FUNCTION_BLOCK FB_Stan_Held EXTENDS FB_SITP_Element
VAR

END_VAR

METHOD FB_init : BOOL
VAR_INPUT
	bInitRetains : BOOL; // if TRUE, the retain variables are initialized (warm start / cold start)
	bInCopyCode : BOOL;  // if TRUE, the instance afterwards gets moved into the copy code (online change)
END_VAR
THIS^.PrzypiszTekstDo (refstEtykieta := THIS^.stNazwa, eJezyk := B_Baza.E_Jezyki.pl, wsTekst	:= "Przerywanie");
THIS^.PrzypiszTekstDo (refstEtykieta := THIS^.stNazwa, eJezyk := B_Baza.E_Jezyki.de, wsTekst	:= "Abbruch");    
THIS^.PrzypiszTekstDo (refstEtykieta := THIS^.stNazwa, eJezyk := B_Baza.E_Jezyki.en, wsTekst	:= "Aborting");
END_METHOD

METHOD PUBLIC WywolajAkcjePBDlaStanu : BOOL
VAR_INPUT
	iNumerPB				: INT;
END_VAR
WywolajAkcjePBDlaStanu			:= THIS^.refstDaneSITP.refarrPB [iNumerPB].SP_Held ();
END_METHOD

(*			
	EVERDE sp. z o.o.
	Rafał Osajda		18.06.2025		TC 4024.66
	Zwraca true jak wyjście ze stanu jest możliwe
*)
METHOD PUBLIC ZwrocCzyMoznaWyjscZeStanu : BOOL
//warunki wyjść dla każdego ze stanów osobnym FB
IF (THIS^.refstDaneSITP.ePolecenieZmianyStanu = E_SITP_PolecenieZmianyStanu.Abort) THEN
	IF (THIS^.refstDaneSITP.arrStanyWlaczoneWTrybie [B_Baza.E_StanyPracy.Aborting]) THEN
		ZwrocCzyMoznaWyjscZeStanu					:= THIS^.ZgodaNaZmianeStanu (B_Baza.E_StanyPracy.Aborting);
	ELSE
		ZwrocCzyMoznaWyjscZeStanu					:= THIS^.BrakZgodyNaZmieneStanu (2);	//Stan do którego chcemy przejść jest wylaczony
	END_IF
ELSIF (THIS^.refstDaneSITP.ePolecenieZmianyStanu = E_SITP_PolecenieZmianyStanu.Stop) THEN
	IF (THIS^.refstDaneSITP.arrStanyWlaczoneWTrybie [B_Baza.E_StanyPracy.Stopping]) THEN
		ZwrocCzyMoznaWyjscZeStanu					:= THIS^.ZgodaNaZmianeStanu (B_Baza.E_StanyPracy.Stopping);
	ELSE
		ZwrocCzyMoznaWyjscZeStanu					:= THIS^.BrakZgodyNaZmieneStanu (2);	//Stan do którego chcemy przejść jest wylaczony
	END_IF
ELSIF (THIS^.refstDaneSITP.ePolecenieZmianyStanu = E_SITP_PolecenieZmianyStanu.Unhold OR
		(THIS^.refstDaneSITP.refbZredukowanaLiczbaPrzyciskow AND THIS^.refstDaneSITP.ePolecenieZmianyStanu = E_SITP_PolecenieZmianyStanu.Start)) THEN
	IF (THIS^.refstDaneSITP.arrStanyWlaczoneWTrybie [B_Baza.E_StanyPracy.Unholding]) THEN
		ZwrocCzyMoznaWyjscZeStanu					:= THIS^.ZgodaNaZmianeStanu (B_Baza.E_StanyPracy.Unholding);
	ELSE
		ZwrocCzyMoznaWyjscZeStanu					:= THIS^.BrakZgodyNaZmieneStanu (2);	//Stan do którego chcemy przejść jest wylaczony
	END_IF
ELSE
	ZwrocCzyMoznaWyjscZeStanu						:= THIS^.BrakZgodyNaZmieneStanu (1);	//Bledny rozkaz dla zmiany stanu
END_IF
END_METHOD

END_FUNCTION_BLOCK

(* stored: Version 1.1.0.1
   POU FB_Stan_Held: Id {b8356b78-e894-020c-3c39-8506fca8dce6}, SpecialFunc None
   Method FB_init: Id {f0715bac-14a5-0d18-1ac0-1bd40aa95a64}
   Method WywolajAkcjePBDlaStanu: Id {bc691794-2656-0fbf-04c0-725b81f33db0}
   Method ZwrocCzyMoznaWyjscZeStanu: Id {9b081693-6bfd-0ce4-0bf2-af9637733dcc} *)
